ABB RobotStudio station: myStat_3.rsstn

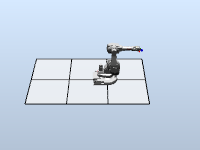
Station myStat_3 (saved by RobotStudio format 3)
Controller Sistema1
  mechanical unit ROB_1: IRB1600_6_120__02, 6 joints, base frame (0, 0, 0) mm
Layout (positions relative to the parent item):
  - IRB1600_6_120__02 [mechanism, from Robots\IRB1600_6_120_G_02.rslib] at (0, 0, 0) mm; joint values [0, 0, 0, 0, 0.5236, 0] (rad or m)
Targets, tools, work objects and paths stored in the station, written as RAPID:
! task T_ROB1
MODULE MainModule
  VAR robtarget positionN:=[[0,0,0],[1,0,0,0],[0,0,0,0],[9E9,9E9,9E9,9E9,9E9,9E9]];
  PROC main()
  ENDPROC
  PROC positioning()
  ENDPROC
  PROC connectSocket()
  ENDPROC
  PROC finalize()
  ENDPROC
  PROC waitConnection()
  ENDPROC
  PROC waitOrders()
  ENDPROC
ENDMODULE

